TYPE TcoEq2Transfer_Control EXTENDS TcoCore.TcoStruct:
STRUCT

	
		
END_STRUCT
END_TYPE

(* stored: Version 1.1.0.1
   DUT TcoEq2Transfer_Control: Id {c28a45ee-88b7-4214-8996-a935e4c98d44} *)
